// SIMATIC S7-200 SMART project (STEP 7-Micro/WIN SMART), CPU ST40

SYMBOL_TABLE Table 1
Start_SW         I0.0
Stop_SW          I0.1
Memory           M0.0
RED              Q0.0
GREEN            Q0.2
RED_Timer        T101
Yellow_Timer     T102
GREEN_Timer      T103
YELLOW           Q0.1
END_SYMBOL_TABLE

ORGANIZATION_BLOCK MAIN:OB1
TITLE=Program Comments
BEGIN
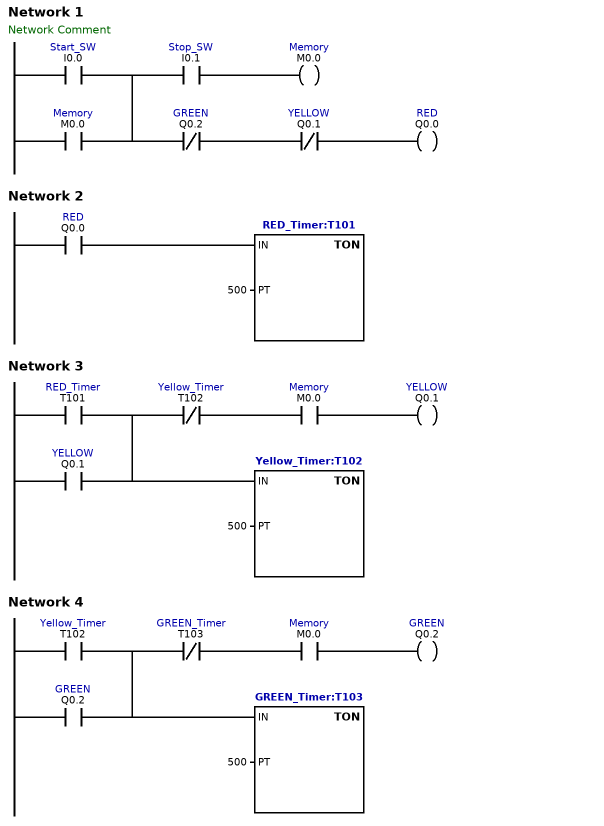
Network 1
// Network Comment
LD     Start_SW:I0.0
O      Memory:M0.0
LPS
A      Stop_SW:I0.1
=      Memory:M0.0
LPP
AN     GREEN:Q0.2
AN     YELLOW:Q0.1
=      RED:Q0.0
Network 2
LD     RED:Q0.0
TON    RED_Timer:T101, 500
Network 3
LD     RED_Timer:T101
O      YELLOW:Q0.1
LPS
AN     Yellow_Timer:T102
A      Memory:M0.0
=      YELLOW:Q0.1
LPP
TON    Yellow_Timer:T102, 500
Network 4
// (network saved uncompiled; LAD cells follow)
// row 0: c0 -| |- Yellow_Timer:T102 v  c1 -|/|- GREEN_Timer:T103  c2 -| |- Memory:M0.0  c3 -( ) GREEN:Q0.2
// row 1: c0 -| |- GREEN:Q0.2 ^  c1 --  c2 [TON GREEN_Timer:T103 IN:=power@row1, PT:=500]
// row 2: c2 [box]
END_ORGANIZATION_BLOCK
